(*	| author		| Beckhoff Automation Poland	|	*)
(* 	-------------------------------------------------	*)
(*	| wersion		| 1.0							|	*)
(* 	-------------------------------------------------	*)
(*	| TC version	| 3.1.4024.7					| 	*)
(* 	-------------------------------------------------	*)
(*	| date			| 19.05.2020					|	*)
(* 	-------------------------------------------------	*)
(*	| description	| custom keypad with hotkeys	|  	*)

PROGRAM MAIN
VAR
	iTest 	: INT;
	sTest	: STRING;
END_VAR

END_PROGRAM

(* stored: Version 1.1.0.1, ProductVersion 3.1.4024.3
   POU MAIN: Id {618e2290-6191-469e-bbb1-e120615f54a4}, SpecialFunc None *)
